// TwinCAT 3 PLC project EL2008Led
// ProgramVersion: 3.1.4026.9
// libraries:
//   Tc2_Standard, * (Beckhoff Automation GmbH)
//   Tc2_System, * (Beckhoff Automation GmbH)
// project tree:
//   DUTs/ E_Color.TcDUT
//   / PlcTask.TcTTO
//   POUs/ MAIN.TcPOU
// real-time tasks:
//   TASK PlcTask: cycle T#10ms, priority 20, ADS port 350
// I/O:
//   DEVICE デバイス 2 (EtherCAT), AmsNetId 169.254.163.179.3.1
//     ターミナル 1 (EK1100) [EK1100 EtherCAT Coupler (2A E-Bus)]
//       ターミナル 2 (EL9410) [EL9410 E-Bus Power Supplier  (Diagnostics)]
//       ターミナル 3 (EL2008) [EL2008 8Ch. Dig. Output 24V, 0.5A]
//       ターミナル 4 (EL2008) [EL2008 8Ch. Dig. Output 24V, 0.5A]
//       ターミナル 9 (EL9011) [EL9011 End Terminal]
//     ターミナル 5 (EK1100) [EK1100 EtherCAT Coupler (2A E-Bus)]
//       ターミナル 6 (EL2004) [EL2004 4Ch. Dig. Output 24V, 0.5A]
//       ターミナル 10 (EL9011) [EL9011 End Terminal]
//     ターミナル 7 (EK1100) [EK1100 EtherCAT Coupler (2A E-Bus)]
//       ターミナル 8 (EL3318) [EL3318 8Ch. Ana Input Thermocouple (TC)]
//       ターミナル 11 (EL9011) [EL9011 End Terminal]
// variable links:
//   (this object) <-> Device 2 (EtherCAT)/Term 1 (EK1100)/Term 3 (EL2008)
//     PlcTask Outputs/MAIN.bLed1[0] <-> Channel 1/Output
//     PlcTask Outputs/MAIN.bLed1[1] <-> Channel 3/Output
//     PlcTask Outputs/MAIN.bLed1[2] <-> Channel 5/Output
//     PlcTask Outputs/MAIN.bLed1[3] <-> Channel 7/Output
//     PlcTask Outputs/MAIN.bLed2[0] <-> Channel 2/Output
//     PlcTask Outputs/MAIN.bLed2[1] <-> Channel 4/Output
//     PlcTask Outputs/MAIN.bLed2[2] <-> Channel 6/Output
//     PlcTask Outputs/MAIN.bLed2[3] <-> Channel 8/Output
//   (this object) <-> Device 2 (EtherCAT)/Term 1 (EK1100)/Term 4 (EL2008)
//     PlcTask Outputs/MAIN.bLed1[0] <-> Channel 1/Output
//     PlcTask Outputs/MAIN.bLed1[1] <-> Channel 3/Output
//     PlcTask Outputs/MAIN.bLed1[2] <-> Channel 5/Output
//     PlcTask Outputs/MAIN.bLed1[3] <-> Channel 7/Output
//     PlcTask Outputs/MAIN.bLed2[0] <-> Channel 2/Output
//     PlcTask Outputs/MAIN.bLed2[1] <-> Channel 4/Output
//     PlcTask Outputs/MAIN.bLed2[2] <-> Channel 6/Output
//     PlcTask Outputs/MAIN.bLed2[3] <-> Channel 8/Output

CONFIGURATION EL2008Led
    RESOURCE PLC ON TwinCAT3
        TASK PlcTask(INTERVAL := T#10ms, PRIORITY := 20);
        PROGRAM MAIN WITH PlcTask : MAIN;
    END_RESOURCE
END_CONFIGURATION

// ---- DUTs/E_Color.TcDUT
{attribute 'qualified_only'}
{attribute 'strict'}
{attribute 'to_string'}
TYPE E_Color :
(
	eRed,
	eYellow,
	eGreen,
	eWhite
)INT;
END_TYPE

// ---- POUs/MAIN.TcPOU
PROGRAM MAIN
VAR
	eLedColor		:E_Color;
	bLed1			:ARRAY[E_Color.eRed..E_Color.eWhite] OF BOOL;
	bLed2			:ARRAY[E_Color.eRed..E_Color.eWhite] OF BOOL;
	
	i				:INT;
END_VAR

i:=i+1;

IF i=10 THEN
	bLed1[E_Color.eRed]:=TRUE;
ELSIF i=20 THEN
	bLed1[E_Color.eYellow]:=TRUE;
ELSIF i=30 THEN
	bLed1[E_Color.eGreen]:=TRUE;
ELSIF i=40 THEN
	bLed1[E_Color.eWhite]:=TRUE;
ELSIF i=50 THEN
	bLed2[E_Color.eRed]:=TRUE;
ELSIF i=60 THEN
	bLed2[E_Color.eYellow]:=TRUE;
ELSIF i=70 THEN
	bLed2[E_Color.eGreen]:=TRUE;
ELSIF i=80 THEN
	bLed2[E_Color.eWhite]:=TRUE;
ELSIF i=100 THEN
	FOR eLedColor:= E_Color.eRed TO E_Color.eWhite DO
		bLed1[eLedColor]:=FALSE;
		bLed2[eLedColor]:=FALSE;
	END_FOR
END_IF

END_PROGRAM
